INTERFACE I_INT EXTENDS I_Datatype

PROPERTY PUBLIC Value : REFERENCE TO INT
GET
END_GET
END_PROPERTY

END_INTERFACE

(* stored: Version 1.1.0.1, ProductVersion 3.1.4024.15
   Itf I_INT: Id {0d55eed5-df3f-0f64-035c-fe3e51fefa5b}
   Property Value: Id {b7035116-cb04-0859-323f-0056b1ec550e}
   Get Get: Id {3dd1c3fc-f5be-0191-08c2-4e1b3d28b6ca} *)
